Staubli VAL3: AfterArrayCut.pgx

public program AfterArrayCut(num x_nWorkplaceIn, num x_nTrajIndex)
begin
  //参数：x_nWorkplaceIn 工位序号，传入的参数是 DataBase:nWorkPlaceIndex
  //参数：x_nTrajIndex 路径序号，传入的参数是TxtFile:nReadTrajIndex
  //引用位置:Motion:Move.pgx
  //功能：在阵列之后添加动作,一般是融覆阵列后要发出动作
  //备注：
  //








end
